SUBAPPLICATION GreenWhiteBackground_Knickdeichsel_heben (* Subapplication Type *)
  (* Standard: 61499-2 *)
  (* Version 1.0, 2023-02-11, franz *)
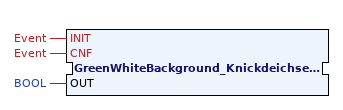
  EVENT_INPUT
    INIT;
    CNF;
  END_EVENT
  VAR_INPUT
    OUT : BOOL;
  END_VAR
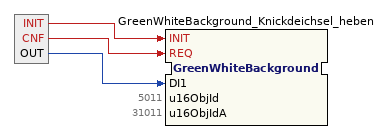
  FBS
    GreenWhiteBackground_Knickdeichsel_heben : GreenWhiteBackground(u16ObjId := 5011, u16ObjIdA := 31011);
  END_FBS
  EVENT_CONNECTIONS
    INIT TO GreenWhiteBackground_Knickdeichsel_heben.INIT;
    CNF TO GreenWhiteBackground_Knickdeichsel_heben.REQ;
  END_CONNECTIONS
  DATA_CONNECTIONS
    OUT TO GreenWhiteBackground_Knickdeichsel_heben.DI1;
  END_CONNECTIONS
END_SUBAPPLICATION
